// TwinCAT 3 PLC project Test_Actuator
// Company: RafalOS
// ProgramVersion: 3.1.4024.0
// libraries:
//   Tc2_Standard, * (Beckhoff Automation GmbH)
//   Tc2_System, * (Beckhoff Automation GmbH)
//   Tc3_Module, * (Beckhoff Automation GmbH)
//   TcUnit, * (www.tcunit.org)
// project tree:
//   / PlcTask.TcTTO
//   TESTs/ PRG_Test.TcPOU
// real-time tasks:
//   TASK PlcTask: cycle T#10ms, priority 20, ADS port 350

CONFIGURATION Test_Actuator
    RESOURCE PLC ON TwinCAT3
        TASK PlcTask(INTERVAL := T#10ms, PRIORITY := 20);
        PROGRAM PRG_Test WITH PlcTask : PRG_Test;
    END_RESOURCE
END_CONFIGURATION

// ---- TESTs/PRG_Test.TcPOU
PROGRAM PRG_Test
VAR
END_VAR


	TcUnit.RUN_IN_SEQUENCE ();

END_PROGRAM
